// TIA Portal V20 export
TYPE "LWONIK_typeRollChangeMode"
// stored: Access Published
   STRUCT
      Auto : Bool;
      RollChange : Bool;
   END_STRUCT;
END_TYPE
